Fanuc KAREL source: kt00134.KL

-- PROVISIONAL review KL for V940-1; original PC SHA256 b3f2fdebe0c034315d3e12f065ff1d4e3bd64d0deb66644975edec8145f67975
-- Incomplete behavior may be omitted. Consult companion uncertainty JSON. Do not deploy.
PROGRAM KT00134
%NOLOCKGROUP
VAR
  I1 : INTEGER
  OUT : REAL
-- UNRESOLVED_DECL Y2 type=002018
BEGIN
  -- V9_ZERO_TABLE_METADATA_HINT layout=0001; no indexed target words; source/name/runtime held
  -- UNRESOLVED_PC offsets 5-16; opcodes 2E,23
  -- UNRESOLVED_PC offsets 21-35; opcodes 2E,22,9D,33,B2
  -- UNRESOLVED_PC offsets 40-63; opcodes 21,22,9D,33,B1,55,64,23
  -- UNRESOLVED_PC offsets 68-72; opcodes 7F
END KT00134
